Staubli VAL3: makeMaxSizeList.pgx

program makeMaxSizeList(num& x_nResult[])
  local string l_sPalletName
  local num l_nSize
  local num i
  local num l_nSizePallet[4]
  local string l_sTemp
  local string l_sEmpty
begin
  //
  // INIT
  //
  sPalletName=""
  // make the list of the max size list of pallet
  call pallet:getSize(l_nSize)
  resize(sPalletName,1,max(1,l_nSize))
  resize(nMax,1,max(1,l_nSize))
  //
  // build the list
  //
  for i=0 to l_nSize-1
    call pallet:get(l_sPalletName,i)
    if l_sPalletName!=""
      call pallet:getSizePallet(l_sPalletName,l_nSizePallet)
      nMax[i]=l_nSizePallet
      sPalletName[i]=l_sPalletName
    endIf
  endFor
end
